(*********************************** G.D S.p.A. - Technical Department ***********************************
============= PROGRAM INFO ============
FOLDER:             TBD
MACHINES INVOLVED:  TBD 

============= DESCRIPTION =============
csp main interface program

============= REVISIONS ===============
Date		Version	 	Author      	Description             
----------	-------		------------  	--------------------------------------------
2019/09/27 	0000.00	 	M.Grasso		Creation of the PRG

**********************************************************************************************************)
PROGRAM _csp_case_topRail_normal
VAR
END_VAR

(* CASE *)
	(* TOP RAIL *)
		(* ACC-U-CHANGE *)
		csp_case_topRail_accU();

END_PROGRAM

(* stored: Version 1.1.0.1, ProductVersion 3.1.4024.3
   POU _csp_case_topRail_normal: Id {af697e85-27cc-4b01-a3b0-53aa3571853b}, SpecialFunc None *)
